(* IEC 61131-3 sources: Std_PalletMover/Class/HandleSteeringCurtisAC2F, 1 file *)

(* ---- HandleSteeringCurtisAC2F.st ---- *)
#define AUTOTIMERLIMIT 3 SEC

(*!
<Class
	Name               = "HandleSteeringCurtisAC2F"
	Revision           = "0.0"
	RealtimeTask       = "false"
	CyclicTask         = "true"
	BackgroundTask     = "false"
	Sigmatek           = "false"
	OSInterface        = "false"
	HighPriority       = "false"
	Automatic          = "false"
	UpdateMode         = "Prescan"
	SharedCommandTable = "true"
	Objectsize         = "(630,120)">
	<Channels>
		<Server Name="CorrectedActual" Visualized="false" Initialize="false" WriteProtected="true" Retentive="false"/>
		<Server Name="ReferenceOffset" Visualized="false" Initialize="false" WriteProtected="false" Retentive="SRam"/>
		<Server Name="ScalingFactor" Visualized="false" Initialize="true" WriteProtected="false" Retentive="File" Comment="Scaling factor between local setpoint/actual and drive setpoint/actual.&#13;&#10;&#13;&#10;PLC Setpoint * ScalingFactor = Drive Setpoint&#13;&#10;Drive Actual / ScalingFactor = PLC Actual"/>
		<Server Name="STARTREF" Visualized="false" Initialize="false" WriteProtected="false" Retentive="false"/>
		<Client Name="ActualRaw" Required="true" Internal="false"/>
		<Client Name="objCurtisAC2F" Required="true" Internal="false"/>
		<Client Name="SafetyEncoderValue" Required="true" Internal="false"/>
		<Client Name="SetpointRaw" Required="true" Internal="false"/>
	</Channels>
	<Network Name="HandleSteeringCurtisAC2F">
		<!-- List of Components in this network -->
		<Components>
			<Object
				Name       = "_base"
				Class      = "HandleSteering"
				Position   = "(218,120)"
				Visualized = "false">
				<Channels>
					<Server Name="Actual"/>
					<Server Name="BusyReferencing"/>
					<Server Name="ClassSvr"/>
					<Server Name="IsReferenced"/>
					<Server Name="Setpoint"/>
				</Channels>
			</Object>
		</Components>
		<Comments>
		</Comments>
		<!-- List of Connections in this network -->
		<Connections>
			<Connection Source="this.ClassSvr" Destination="_base.ClassSvr" Vertices="(968,210),(796,210),"/>
			<Connection Source="this.Actual" Destination="_base.Actual" Vertices="(968,330),(796,330),"/>
			<Connection Source="this.Setpoint" Destination="_base.Setpoint" Vertices="(968,270),(796,270),"/>
			<Connection Source="this.IsReferenced" Destination="_base.IsReferenced" Vertices="(968,390),(796,390),"/>
			<Connection Source="this.BusyReferencing" Destination="_base.BusyReferencing" Vertices="(968,450),(796,450),"/>
		</Connections>
		<!-- Headerfiles -->
		<Options>
		</Options>
	</Network>
</Class>
*)
#pragma using HandleSteering

HandleSteeringCurtisAC2F : CLASS
: HandleSteering
  //Servers:
	ReferenceOffset 	: SvrCh_REAL;
	CorrectedActual 	: SvrCh_REAL;
	ScalingFactor 	: SvrCh_REAL;
	STARTREF 	: SvrCh_DINT;
  //Clients:
	objCurtisAC2F 	: CltChCmd_Curtis_AC2F;
	SafetyEncoderValue 	: CltCh_REAL;
	ActualRaw 	: CltCh_DINT;
	SetpointRaw 	: CltCh_DINT;
  //Variables:
		_initCounter 	: DINT;
		_init 	: DINT;
  //Functions:

	FUNCTION VIRTUAL GLOBAL Init;

	FUNCTION VIRTUAL GLOBAL CyWork
		VAR_INPUT
			EAX 	: UDINT;
		END_VAR
		VAR_OUTPUT
			state (EAX) 	: UDINT := READY;
		END_VAR;

	FUNCTION VIRTUAL GLOBAL GetReferenced
		VAR_OUTPUT
			returnValue 	: DINT;
		END_VAR;

	FUNCTION VIRTUAL GLOBAL GetDriveStatus
		VAR_OUTPUT
			returnValue 	: tDriveStatus;
		END_VAR;

	FUNCTION VIRTUAL _forwardSetpoint
		VAR_INPUT
			inputSetpoint 	: REAL;
		END_VAR;

	FUNCTION VIRTUAL _getActual
		VAR_OUTPUT
			returnValue 	: REAL;
		END_VAR;

	FUNCTION VIRTUAL GLOBAL StartReferencing;

	FUNCTION _readClients;

	FUNCTION VIRTUAL GLOBAL STARTREF::Write
		VAR_INPUT
			input (EAX) 	: DINT;
		END_VAR
		VAR_OUTPUT
			result (EAX) 	: DINT;
		END_VAR;
  //Tables:
	FUNCTION @STD
		VAR_OUTPUT
			ret_code	: CONFSTATES;
		END_VAR;
	FUNCTION GLOBAL TAB @CT_;
END_CLASS;

#pragma usingLtd Curtis_AC2F

FUNCTION VIRTUAL GLOBAL HandleSteeringCurtisAC2F::Init
  _initCounter += 1;

  if (_initCounter = 10) then
    _init := TRUE;
  end_if;

END_FUNCTION

FUNCTION VIRTUAL GLOBAL HandleSteeringCurtisAC2F::GetDriveStatus
	VAR_OUTPUT
		returnValue 	: tDriveStatus;
	END_VAR
  VAR
  	tmpDriveMode  : Curtis_Base::eCurtisDriveMode;
  END_VAR

  tmpDriveMode := objCurtisAC2F.DriveMode.Read();

  if tmpDriveMode = Curtis_Base::cdm_Auto then
    returnValue.ds_DriveMode := HandleSteering::dm_Auto;
  elsif tmpDriveMode = Curtis_Base::cdm_Manual then
    returnValue.ds_DriveMode := HandleSteering::dm_Manual;
  elsif tmpDriveMode = Curtis_Base::cdm_Referencing then
    returnValue.ds_DriveMode := HandleSteering::dm_Referencing;
  elsif tmpDriveMode = Curtis_Base::cdm_EmergencyStop then
    returnValue.ds_DriveMode := HandleSteering::dm_EmergencyStop;
  else
    returnValue.ds_DriveMode := HandleSteering::dm_Idle;
  end_if;

  returnValue.ds_Referenced := objCurtisAC2F.Referenced.Read();
  returnValue.ds_Setpoint := SetpointRaw.Read();
  returnValue.ds_Actual := _getActual();
  returnValue.ds_FaultCode := objCurtisAC2F.FaultCode.Read();
  returnValue.ds_CommunicationOK := objCurtisAC2F.CommunicationOk.Read();
  returnValue.ds_EstopOK := objCurtisAC2F.EmStopOk;

END_FUNCTION

FUNCTION VIRTUAL HandleSteeringCurtisAC2F::_forwardSetpoint
	VAR_INPUT
		inputSetpoint 	: REAL;
	END_VAR
  VAR
  	tempSet : REAL;
  END_VAR

  tempSet := ScalingFactor * (inputSetpoint - ReferenceOffset);
  SetpointRaw.Write(to_dint(tempSet));

END_FUNCTION

FUNCTION VIRTUAL GLOBAL HandleSteeringCurtisAC2F::CyWork
	VAR_INPUT
		EAX 	: UDINT;
	END_VAR
	VAR_OUTPUT
		state (EAX) 	: UDINT;(* := READY *)
	END_VAR

  _readClients();

  if _init = TRUE & SafetyEncoderValue <> 0 then
    //StartReferencing();
     ReferenceOffset.Write(input:=SafetyEncoderValue.Read());
    _init := FALSE;
    IsReferenced := TRUE;
  end_if;

  if BusyReferencing = TRUE then
    if ActualRaw <> 0 | objCurtisAC2F.BusyReferencing = FALSE then
      objCurtisAC2F.StartReferencing();
    end_if;

    if objCurtisAC2F.BusyReferencing = 1 & BusyReferencing = TRUE then
      if objCurtisAC2F.Referenced = 1 & objCurtisAc2F.EncoderValue = 0 then
        if ReferenceOffset <> SafetyEncoderValue.Read() then
          ReferenceOffset.Write(input:=SafetyEncoderValue.Read());
        end_if;
        objCurtisAC2F.StopReferencing();
        BusyReferencing := FALSE;
        IsReferenced := TRUE;
      end_if;
    end_if;
  end_if;

  Actual := to_real(ActualRaw)/ScalingFactor;
  CorrectedActual := Actual + ReferenceOffset;

END_FUNCTION

FUNCTION VIRTUAL HandleSteeringCurtisAC2F::_getActual
	VAR_OUTPUT
		returnValue 	: REAL;
	END_VAR

  if IsReferenced = TRUE | BusyReferencing = FALSE then
    returnValue := CorrectedActual;
  else
    returnValue := 0;
  end_if;

END_FUNCTION

FUNCTION VIRTUAL GLOBAL HandleSteeringCurtisAC2F::StartReferencing

  BusyReferencing := TRUE;
  IsReferenced := FALSE;

END_FUNCTION

FUNCTION VIRTUAL GLOBAL HandleSteeringCurtisAC2F::STARTREF::Write
	VAR_INPUT
		input (EAX) 	: DINT;
	END_VAR
	VAR_OUTPUT
		result (EAX) 	: DINT;
	END_VAR

	STARTREF := input;
  if STARTREF = 1 then
    StartReferencing();
  end_if;
	result := STARTREF;

END_FUNCTION

FUNCTION HandleSteeringCurtisAC2F::_readClients

  SafetyEncoderValue := SafetyEncoderValue.Read();
  ActualRaw := ActualRaw.Read();
  SetpointRaw := SetpointRaw.Read();

END_FUNCTION

FUNCTION VIRTUAL GLOBAL HandleSteeringCurtisAC2F::GetReferenced
	VAR_OUTPUT
		returnValue 	: DINT;
	END_VAR

  returnValue := objCurtisAC2F.Referenced;

END_FUNCTION
